TYPE MediatorGroupStatus :
STRUCT
	Valid          			: BOOL;
    Busy           			: BOOL;
    GroupMoving    			: BOOL;
    GroupHoming    			: BOOL;
    GroupErrorStop 			: BOOL;
    GroupNotReady  			: BOOL;
    GroupStandby   			: BOOL;
    GroupStopping  			: BOOL;
    GroupDisabled  			: BOOL;
    AllAxesStanding			: BOOL;
    InPosition     			: BOOL;
    Error          			: BOOL;
    ErrorId        			: UDINT;
	// custom statuses for this application
	Enabled					: BOOL;
END_STRUCT
END_TYPE

(* stored: Version 1.1.0.1, ProductVersion 3.1.4024.12
   DUT MediatorGroupStatus: Id {32999573-d701-00d8-1ee2-09643aad92ba} *)
